PROGRAM P_TableVacuum
VAR
	FB_TableVacuum:ARRAY[1..number_TableVacuum] OF FB_TableVacuum;
	i:INT;	
	log_ErrorEnum:TabVacErrorEnum;
	log_ID:INT;
END_VAR

ACT_LOG();

FOR i:=1 TO number_TableVacuum DO
	FB_TableVacuum[i](
		vacuum_measured:= GVL_API.stTableVacuum[i].vacuum_measured, 
		vacuum_min:= GVL_API.stTableVacuum[i].vacuum_min, 
		vacuum_max:= GVL_API.stTableVacuum[i].vacuum_max, 
		setpoint:= GVL_API.stTableVacuum[i].setpoint, 
		vacuum_offset_collector:= GVL_API.stTableVacuum[i].vacuum_offset_collector, 
		setpoint_range_pct:= GVL_API.stTableVacuum[i].setpoint_range_pct, 
		vacuum_timeout:= GVL_API.stTableVacuum[i].vacuum_timeout, 
		vacuum_off_timeout:= GVL_API.stTableVacuum[i].vacuum_off_timeout, 
		IO_Error:=P_Modbus_RTU.station_error[1] OR P_Modbus_RTU.station_error[2],
		state=> GVL_API.stTableVacuum[i].state, 
		error_code=> GVL_API.stTableVacuum[i].error_code, 
		Run=> stOutput.bqVacRun[i], 
		error=> GVL_API.stTableVacuum[1].Error, 
		Initialize:= GVL_API.stTableVacuum[i].Initialize, 
		SetVacuumOn:= GVL_API.stTableVacuum[i].SetVacuumOn, 
		SetVacuumOff:= GVL_API.stTableVacuum[i].SetVacuumOff, 
		Setoff:=GVL_API.stTableVacuum[i].Setoff  );
		
END_FOR

ACTION ACT_LOG:
(*************************LOG*******************************************)
log_ID:=300;
//initialize
AlarmActionArray[log_ID+1].AlarmMsg.EN	:=CONCAT('TableVacuum initialize, ',LREAL_TO_STRING(GVL_API.stTableVacuum[1].vacuum_min));
AlarmActionArray[log_ID+1].AlarmMsg.EN	:=CONCAT(AlarmActionArray[log_ID+1].AlarmMsg.EN,', ');
AlarmActionArray[log_ID+1].AlarmMsg.EN	:=CONCAT(AlarmActionArray[log_ID+1].AlarmMsg.EN,
																	LREAL_TO_STRING(GVL_API.stTableVacuum[1].vacuum_max));
AlarmActionArray[log_ID+1].AlarmMsg.EN	:=CONCAT(AlarmActionArray[log_ID+1].AlarmMsg.EN,', ');
AlarmActionArray[log_ID+1].AlarmMsg.EN	:=CONCAT(AlarmActionArray[log_ID+1].AlarmMsg.EN,
																	LREAL_TO_STRING(GVL_API.stTableVacuum[1].setpoint_range_pct));														
fbSetAlarm[log_ID+1](
	InUse:=TRUE , 
	EventId:=log_ID+1 , 
	EventActive:=GVL_API.stTableVacuum[1].Initialize , 
	EventClass:=Alm_EventClass.Event , 
	ToTheLogFile:=TRUE, 
	ToTheHistory:=TRUE , 
 );
 //SetVacuumOn
AlarmActionArray[log_ID+2].AlarmMsg.EN	:=CONCAT('TableVacuum SetVacuumOn, ',LREAL_TO_STRING(GVL_API.stTableVacuum[1].setpoint));
AlarmActionArray[log_ID+2].AlarmMsg.EN	:=CONCAT(AlarmActionArray[log_ID+2].AlarmMsg.EN,', ');
AlarmActionArray[log_ID+2].AlarmMsg.EN	:=CONCAT(AlarmActionArray[log_ID+2].AlarmMsg.EN,
																	LREAL_TO_STRING(GVL_API.stTableVacuum[1].vacuum_timeout));

fbSetAlarm[log_ID+2](
	InUse:=TRUE , 
	EventId:=log_ID+2 , 
	EventActive:=GVL_API.stTableVacuum[1].SetVacuumOn , 
	EventClass:=Alm_EventClass.Event , 
	ToTheLogFile:=TRUE, 
	ToTheHistory:=TRUE , 
 );
 //SetVacuumOff
AlarmActionArray[log_ID+3].AlarmMsg.EN	:=CONCAT('TableVacuum SetVacuumOff, ',LREAL_TO_STRING(GVL_API.stTableVacuum[1].vacuum_off_timeout));

fbSetAlarm[log_ID+3](
	InUse:=TRUE , 
	EventId:=log_ID+3 , 
	EventActive:=GVL_API.stTableVacuum[1].SetVacuumOff , 
	EventClass:=Alm_EventClass.Event , 
	ToTheLogFile:=TRUE, 
	ToTheHistory:=TRUE , 
 );

//ERROR,log_ErrorEnum只能等于一个常数
CASE GVL_API.stTableVacuum[1].error_code  OF
0	:	log_ErrorEnum	:=	0	;
1	:	log_ErrorEnum	:=	1	;
2	:	log_ErrorEnum	:=	2	;
3	:	log_ErrorEnum	:=	3	;
4	:	log_ErrorEnum	:=	4	;
5	:	log_ErrorEnum	:=	5	;
6	:	log_ErrorEnum	:=	6	;
7	:	log_ErrorEnum	:=	7	;
8	:	log_ErrorEnum	:=	8	;
666	:	log_ErrorEnum	:=	666	;


END_CASE

AlarmActionArray[log_ID+9].AlarmMsg.EN	:=CONCAT('TableVacuum Error: ',TO_STRING(log_ErrorEnum));
fbSetAlarm[log_ID+9](
	InUse:=TRUE , 
	EventId:=log_ID+9 , 
	EventActive:=GVL_API.stTableVacuum[1].error_code<>0 AND GVL_API.stTableVacuum[1].error_code<>666   , 
	EventClass:=Alm_EventClass.Alarm , 
	ToTheLogFile:=TRUE, 
	ToTheHistory:=TRUE , 
 );
 
//reset
AlarmActionArray[log_ID+10].AlarmMsg.EN	:=	'TableVacuum Reset ';
fbSetAlarm[log_ID+10](
	InUse:=TRUE , 
	EventId:=log_ID+10 , 
	EventActive:=GVL_API.stTableVacuum[1].Setoff  , 
	EventClass:=Alm_EventClass.Event , 
	ToTheLogFile:=TRUE, 
	ToTheHistory:=TRUE , 
 );
END_ACTION

END_PROGRAM

(* stored: Version 1.1.0.1, ProductVersion 3.1.4024.11
   POU P_TableVacuum: Id {43f8e08a-f449-4e55-a578-cf3e5d808385}, SpecialFunc None
   Action ACT_LOG: Id {d25b0494-a922-4a4a-bb34-0e4e18a05aa0} *)
